RoboDK station: TM5-900 Workstation.rdk

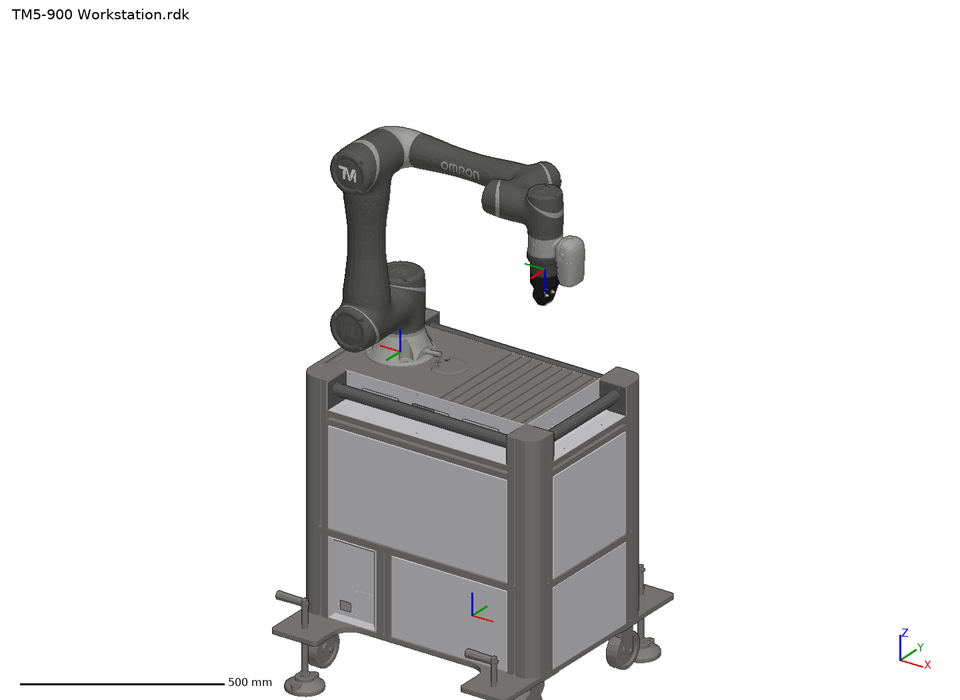
[picture v0: the station drawn from its stored meshes, robots at their saved joint values, targets as dots, program paths as lines]
Station TM5-900 Workstation (saved by RoboDK 5.3.5). Poses are relative to the parent item; angles as X-Y-Z fixed-axis rotations.
  - frame TM5-900 Workstation at (0, 2000, 0) mm
    - frame Omron TM5-900 Base at (-215, 0, 658) mm, rotated rx 0 ry 0 rz 180 deg
      - robot Omron TM5-900: 6 axes, payload 4 kg, reach 900 mm, repeatability 0.1 mm, weight 30 kg
          modified DH rows (alpha deg, a mm, theta deg, d mm): 0, 0, 0, 145.2; 90, 0, 90, 0; 0, 429, 0, 0; 0, 411, -90, 122.3; -90, 0, 0, 106.5; 90, 0, 180, 114.15
          joint limits [-270, -180, -155, -180, -180, -270] to [270, 180, 155, 180, 180, 270]; home [0, 0, 90, -90, 90, 0]; saved at [180, 0, 90, 0, 90, 0]
        - tool RobotiQ Coupler v2, TCP at (0, 0, 20) mm, size 123 x 75 x 16.9 mm, geometry from RobotiQ Coupler v2.step
        - tool Force Sensor v2, TCP at (0, 0, 200) mm, size 89 x 136.8 x 41.5 mm, geometry from Force Sensor v2.step
        - frame RobotiQ 2F85 Base at (0, 0, 42.8) mm, rotated rx 0 ry 0 rz 180 deg
          - robot RobotiQ 2F85: 1 axes, payload 5 kg
              joint limits [0] to [85]; home [85]; saved at [85]
    - object MOBILE_WORKSTATION v4 at (0, 0, 0) mm, size 713 x 729 x 812 mm, geometry from MOBILE_WORKSTATION v4.step
